(* CoDeSys 2.3 export: 6SHU-P2_V2.EXP *)

(* POU MAIN, CFC *)
PROGRAM MAIN
VAR
	TCT: ISTOK_TaskCycleTime;
END_VAR
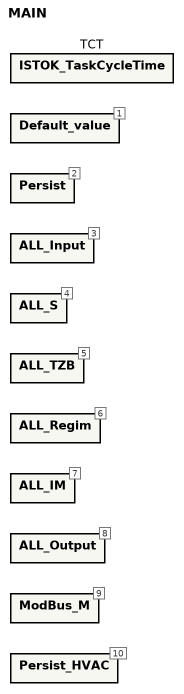
_CFC_ (* Continuous Function Chart, elements in execution order *)
#0 TCT:ISTOK_TaskCycleTime()
#1 Default_value()
#2 Persist()
#3 ALL_Input()
#4 ALL_S()
#5 ALL_TZB()
#6 ALL_Regim()
#7 ALL_IM()
#8 ALL_Output()
#9 ModBus_M()
#10 Persist_HVAC()
_END_CFC_
(* the same logic as Structured Text *)
TCT();
Default_value();
Persist();
ALL_Input();
ALL_S();
ALL_TZB();
ALL_Regim();
ALL_IM();
ALL_Output();
ModBus_M();
Persist_HVAC();
END_PROGRAM

(* POU Lib/ISTOK_TaskCycleTime, CFC *)
FUNCTION_BLOCK ISTOK_TaskCycleTime
VAR_INPUT
END_VAR
VAR_OUTPUT
END_VAR
VAR
END_VAR
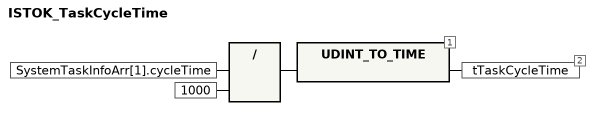
_CFC_ (* Continuous Function Chart, elements in execution order *)
#0 /(SystemTaskInfoArr[1].cycleTime, 1000)
#1 UDINT_TO_TIME(#0)
#2 tTaskCycleTime <= #1
_END_CFC_
END_FUNCTION_BLOCK

(* POU Default_value, CFC *)
PROGRAM Default_value
VAR
END_VAR
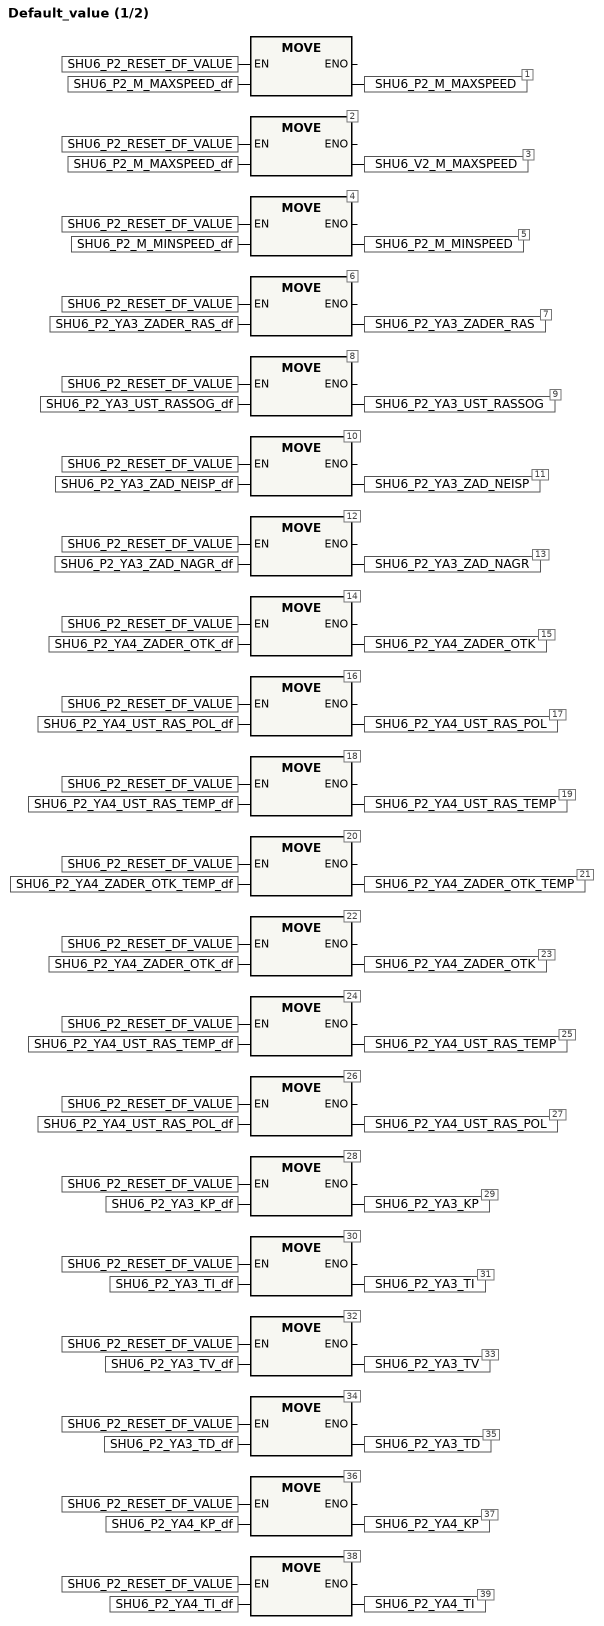
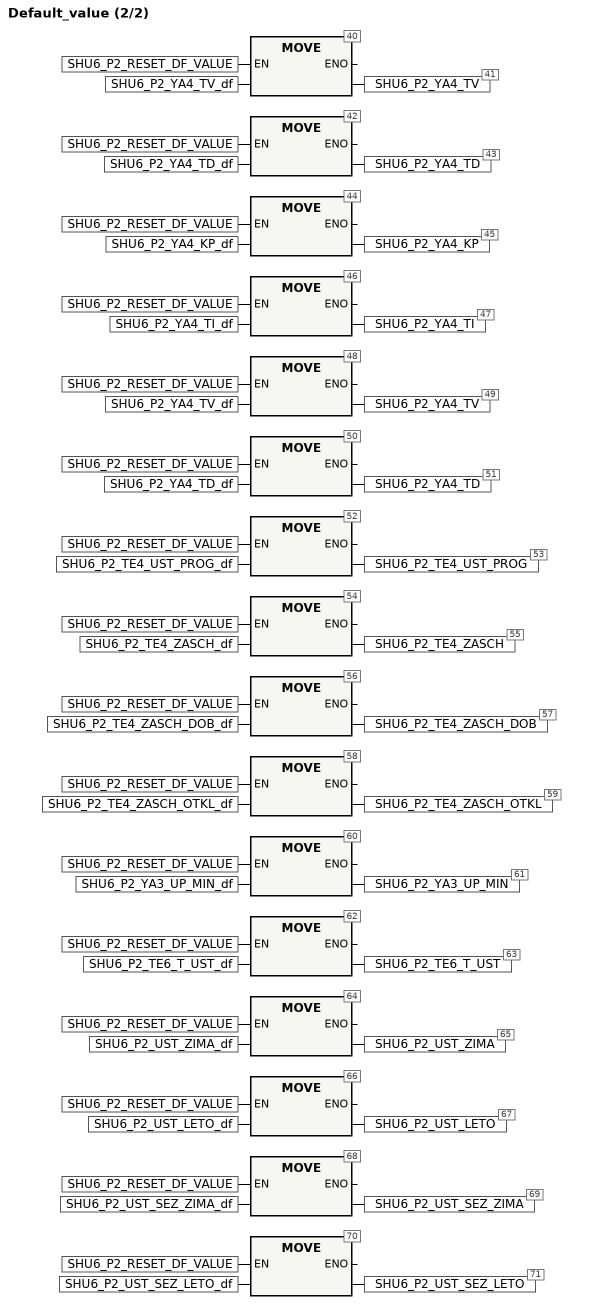
_CFC_ (* Continuous Function Chart, elements in execution order *)
#0 MOVE(EN: SHU6_P2_RESET_DF_VALUE, SHU6_P2_M_MAXSPEED_df)
#1 SHU6_P2_M_MAXSPEED <= #0
#2 MOVE(EN: SHU6_P2_RESET_DF_VALUE, SHU6_P2_M_MAXSPEED_df)
#3 SHU6_V2_M_MAXSPEED <= #2
#4 MOVE(EN: SHU6_P2_RESET_DF_VALUE, SHU6_P2_M_MINSPEED_df)
#5 SHU6_P2_M_MINSPEED <= #4
#6 MOVE(EN: SHU6_P2_RESET_DF_VALUE, SHU6_P2_YA3_ZADER_RAS_df)
#7 SHU6_P2_YA3_ZADER_RAS <= #6
#8 MOVE(EN: SHU6_P2_RESET_DF_VALUE, SHU6_P2_YA3_UST_RASSOG_df)
#9 SHU6_P2_YA3_UST_RASSOG <= #8
#10 MOVE(EN: SHU6_P2_RESET_DF_VALUE, SHU6_P2_YA3_ZAD_NEISP_df)
#11 SHU6_P2_YA3_ZAD_NEISP <= #10
#12 MOVE(EN: SHU6_P2_RESET_DF_VALUE, SHU6_P2_YA3_ZAD_NAGR_df)
#13 SHU6_P2_YA3_ZAD_NAGR <= #12
#14 MOVE(EN: SHU6_P2_RESET_DF_VALUE, SHU6_P2_YA4_ZADER_OTK_df)
#15 SHU6_P2_YA4_ZADER_OTK <= #14
#16 MOVE(EN: SHU6_P2_RESET_DF_VALUE, SHU6_P2_YA4_UST_RAS_POL_df)
#17 SHU6_P2_YA4_UST_RAS_POL <= #16
#18 MOVE(EN: SHU6_P2_RESET_DF_VALUE, SHU6_P2_YA4_UST_RAS_TEMP_df)
#19 SHU6_P2_YA4_UST_RAS_TEMP <= #18
#20 MOVE(EN: SHU6_P2_RESET_DF_VALUE, SHU6_P2_YA4_ZADER_OTK_TEMP_df)
#21 SHU6_P2_YA4_ZADER_OTK_TEMP <= #20
#22 MOVE(EN: SHU6_P2_RESET_DF_VALUE, SHU6_P2_YA4_ZADER_OTK_df)
#23 SHU6_P2_YA4_ZADER_OTK <= #22
#24 MOVE(EN: SHU6_P2_RESET_DF_VALUE, SHU6_P2_YA4_UST_RAS_TEMP_df)
#25 SHU6_P2_YA4_UST_RAS_TEMP <= #24
#26 MOVE(EN: SHU6_P2_RESET_DF_VALUE, SHU6_P2_YA4_UST_RAS_POL_df)
#27 SHU6_P2_YA4_UST_RAS_POL <= #26
#28 MOVE(EN: SHU6_P2_RESET_DF_VALUE, SHU6_P2_YA3_KP_df)
#29 SHU6_P2_YA3_KP <= #28
#30 MOVE(EN: SHU6_P2_RESET_DF_VALUE, SHU6_P2_YA3_TI_df)
#31 SHU6_P2_YA3_TI <= #30
#32 MOVE(EN: SHU6_P2_RESET_DF_VALUE, SHU6_P2_YA3_TV_df)
#33 SHU6_P2_YA3_TV <= #32
#34 MOVE(EN: SHU6_P2_RESET_DF_VALUE, SHU6_P2_YA3_TD_df)
#35 SHU6_P2_YA3_TD <= #34
#36 MOVE(EN: SHU6_P2_RESET_DF_VALUE, SHU6_P2_YA4_KP_df)
#37 SHU6_P2_YA4_KP <= #36
#38 MOVE(EN: SHU6_P2_RESET_DF_VALUE, SHU6_P2_YA4_TI_df)
#39 SHU6_P2_YA4_TI <= #38
#40 MOVE(EN: SHU6_P2_RESET_DF_VALUE, SHU6_P2_YA4_TV_df)
#41 SHU6_P2_YA4_TV <= #40
#42 MOVE(EN: SHU6_P2_RESET_DF_VALUE, SHU6_P2_YA4_TD_df)
#43 SHU6_P2_YA4_TD <= #42
#44 MOVE(EN: SHU6_P2_RESET_DF_VALUE, SHU6_P2_YA4_KP_df)
#45 SHU6_P2_YA4_KP <= #44
#46 MOVE(EN: SHU6_P2_RESET_DF_VALUE, SHU6_P2_YA4_TI_df)
#47 SHU6_P2_YA4_TI <= #46
#48 MOVE(EN: SHU6_P2_RESET_DF_VALUE, SHU6_P2_YA4_TV_df)
#49 SHU6_P2_YA4_TV <= #48
#50 MOVE(EN: SHU6_P2_RESET_DF_VALUE, SHU6_P2_YA4_TD_df)
#51 SHU6_P2_YA4_TD <= #50
#52 MOVE(EN: SHU6_P2_RESET_DF_VALUE, SHU6_P2_TE4_UST_PROG_df)
#53 SHU6_P2_TE4_UST_PROG <= #52
#54 MOVE(EN: SHU6_P2_RESET_DF_VALUE, SHU6_P2_TE4_ZASCH_df)
#55 SHU6_P2_TE4_ZASCH <= #54
#56 MOVE(EN: SHU6_P2_RESET_DF_VALUE, SHU6_P2_TE4_ZASCH_DOB_df)
#57 SHU6_P2_TE4_ZASCH_DOB <= #56
#58 MOVE(EN: SHU6_P2_RESET_DF_VALUE, SHU6_P2_TE4_ZASCH_OTKL_df)
#59 SHU6_P2_TE4_ZASCH_OTKL <= #58
#60 MOVE(EN: SHU6_P2_RESET_DF_VALUE, SHU6_P2_YA3_UP_MIN_df)
#61 SHU6_P2_YA3_UP_MIN <= #60
#62 MOVE(EN: SHU6_P2_RESET_DF_VALUE, SHU6_P2_TE6_T_UST_df)
#63 SHU6_P2_TE6_T_UST <= #62
#64 MOVE(EN: SHU6_P2_RESET_DF_VALUE, SHU6_P2_UST_ZIMA_df)
#65 SHU6_P2_UST_ZIMA <= #64
#66 MOVE(EN: SHU6_P2_RESET_DF_VALUE, SHU6_P2_UST_LETO_df)
#67 SHU6_P2_UST_LETO <= #66
#68 MOVE(EN: SHU6_P2_RESET_DF_VALUE, SHU6_P2_UST_SEZ_ZIMA_df)
#69 SHU6_P2_UST_SEZ_ZIMA <= #68
#70 MOVE(EN: SHU6_P2_RESET_DF_VALUE, SHU6_P2_UST_SEZ_LETO_df)
#71 SHU6_P2_UST_SEZ_LETO <= #70
_END_CFC_
(* the same logic as Structured Text *)
IF SHU6_P2_RESET_DF_VALUE THEN SHU6_P2_M_MAXSPEED := SHU6_P2_M_MAXSPEED_df; END_IF;
IF SHU6_P2_RESET_DF_VALUE THEN SHU6_V2_M_MAXSPEED := SHU6_P2_M_MAXSPEED_df; END_IF;
IF SHU6_P2_RESET_DF_VALUE THEN SHU6_P2_M_MINSPEED := SHU6_P2_M_MINSPEED_df; END_IF;
IF SHU6_P2_RESET_DF_VALUE THEN SHU6_P2_YA3_ZADER_RAS := SHU6_P2_YA3_ZADER_RAS_df; END_IF;
IF SHU6_P2_RESET_DF_VALUE THEN SHU6_P2_YA3_UST_RASSOG := SHU6_P2_YA3_UST_RASSOG_df; END_IF;
IF SHU6_P2_RESET_DF_VALUE THEN SHU6_P2_YA3_ZAD_NEISP := SHU6_P2_YA3_ZAD_NEISP_df; END_IF;
IF SHU6_P2_RESET_DF_VALUE THEN SHU6_P2_YA3_ZAD_NAGR := SHU6_P2_YA3_ZAD_NAGR_df; END_IF;
IF SHU6_P2_RESET_DF_VALUE THEN SHU6_P2_YA4_ZADER_OTK := SHU6_P2_YA4_ZADER_OTK_df; END_IF;
IF SHU6_P2_RESET_DF_VALUE THEN SHU6_P2_YA4_UST_RAS_POL := SHU6_P2_YA4_UST_RAS_POL_df; END_IF;
IF SHU6_P2_RESET_DF_VALUE THEN SHU6_P2_YA4_UST_RAS_TEMP := SHU6_P2_YA4_UST_RAS_TEMP_df; END_IF;
IF SHU6_P2_RESET_DF_VALUE THEN SHU6_P2_YA4_ZADER_OTK_TEMP := SHU6_P2_YA4_ZADER_OTK_TEMP_df; END_IF;
IF SHU6_P2_RESET_DF_VALUE THEN SHU6_P2_YA4_ZADER_OTK := SHU6_P2_YA4_ZADER_OTK_df; END_IF;
IF SHU6_P2_RESET_DF_VALUE THEN SHU6_P2_YA4_UST_RAS_TEMP := SHU6_P2_YA4_UST_RAS_TEMP_df; END_IF;
IF SHU6_P2_RESET_DF_VALUE THEN SHU6_P2_YA4_UST_RAS_POL := SHU6_P2_YA4_UST_RAS_POL_df; END_IF;
IF SHU6_P2_RESET_DF_VALUE THEN SHU6_P2_YA3_KP := SHU6_P2_YA3_KP_df; END_IF;
IF SHU6_P2_RESET_DF_VALUE THEN SHU6_P2_YA3_TI := SHU6_P2_YA3_TI_df; END_IF;
IF SHU6_P2_RESET_DF_VALUE THEN SHU6_P2_YA3_TV := SHU6_P2_YA3_TV_df; END_IF;
IF SHU6_P2_RESET_DF_VALUE THEN SHU6_P2_YA3_TD := SHU6_P2_YA3_TD_df; END_IF;
IF SHU6_P2_RESET_DF_VALUE THEN SHU6_P2_YA4_KP := SHU6_P2_YA4_KP_df; END_IF;
IF SHU6_P2_RESET_DF_VALUE THEN SHU6_P2_YA4_TI := SHU6_P2_YA4_TI_df; END_IF;
IF SHU6_P2_RESET_DF_VALUE THEN SHU6_P2_YA4_TV := SHU6_P2_YA4_TV_df; END_IF;
IF SHU6_P2_RESET_DF_VALUE THEN SHU6_P2_YA4_TD := SHU6_P2_YA4_TD_df; END_IF;
IF SHU6_P2_RESET_DF_VALUE THEN SHU6_P2_YA4_KP := SHU6_P2_YA4_KP_df; END_IF;
IF SHU6_P2_RESET_DF_VALUE THEN SHU6_P2_YA4_TI := SHU6_P2_YA4_TI_df; END_IF;
IF SHU6_P2_RESET_DF_VALUE THEN SHU6_P2_YA4_TV := SHU6_P2_YA4_TV_df; END_IF;
IF SHU6_P2_RESET_DF_VALUE THEN SHU6_P2_YA4_TD := SHU6_P2_YA4_TD_df; END_IF;
IF SHU6_P2_RESET_DF_VALUE THEN SHU6_P2_TE4_UST_PROG := SHU6_P2_TE4_UST_PROG_df; END_IF;
IF SHU6_P2_RESET_DF_VALUE THEN SHU6_P2_TE4_ZASCH := SHU6_P2_TE4_ZASCH_df; END_IF;
IF SHU6_P2_RESET_DF_VALUE THEN SHU6_P2_TE4_ZASCH_DOB := SHU6_P2_TE4_ZASCH_DOB_df; END_IF;
IF SHU6_P2_RESET_DF_VALUE THEN SHU6_P2_TE4_ZASCH_OTKL := SHU6_P2_TE4_ZASCH_OTKL_df; END_IF;
IF SHU6_P2_RESET_DF_VALUE THEN SHU6_P2_YA3_UP_MIN := SHU6_P2_YA3_UP_MIN_df; END_IF;
IF SHU6_P2_RESET_DF_VALUE THEN SHU6_P2_TE6_T_UST := SHU6_P2_TE6_T_UST_df; END_IF;
IF SHU6_P2_RESET_DF_VALUE THEN SHU6_P2_UST_ZIMA := SHU6_P2_UST_ZIMA_df; END_IF;
IF SHU6_P2_RESET_DF_VALUE THEN SHU6_P2_UST_LETO := SHU6_P2_UST_LETO_df; END_IF;
IF SHU6_P2_RESET_DF_VALUE THEN SHU6_P2_UST_SEZ_ZIMA := SHU6_P2_UST_SEZ_ZIMA_df; END_IF;
IF SHU6_P2_RESET_DF_VALUE THEN SHU6_P2_UST_SEZ_LETO := SHU6_P2_UST_SEZ_LETO_df; END_IF;
END_PROGRAM

(* POU Persist, ST *)
PROGRAM Persist
VAR
	Save: WritePersistentData;
END_VAR
Save(NETID:='10.150.4.62.1.1',PORT:=801,START:=TRUE,TMOUT:=t#1s ,BUSY=> ,ERR=> ,	ERRID=> );
Save(NETID:='10.150.4.62.1.1',PORT:=801,START:= FALSE ,TMOUT:=t#1s ,BUSY=> ,ERR=> ,ERRID=> );
END_PROGRAM

(* POU Input/ALL_Input, CFC *)
PROGRAM ALL_Input
VAR
END_VAR
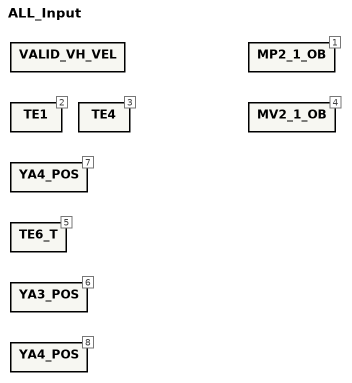
_CFC_ (* Continuous Function Chart, elements in execution order *)
#0 VALID_VH_VEL()
#1 MP2_1_OB()
#2 TE1()
#3 TE4()
#4 MV2_1_OB()
#5 TE6_T()
#6 YA3_POS()
#7 YA4_POS()
#8 YA4_POS()
_END_CFC_
(* the same logic as Structured Text *)
VALID_VH_VEL();
MP2_1_OB();
TE1();
TE4();
MV2_1_OB();
TE6_T();
YA3_POS();
YA4_POS();
YA4_POS();
END_PROGRAM

(* POU Input/VALID_VH_VEL, CFC *)
PROGRAM VALID_VH_VEL
VAR
	SHU6_P2_UST_SEZ_LETO_OLD: REAL;
	SHU6_P2_UST_SEZ_ZIMA_OLD: REAL;

	RT_VKL_OLD_SEZ_LETO: R_TRIG;
	RT_VKL_OLD_SEZ_ZIMA: R_TRIG;

	(*_____________________________________*)
	SHU6_P2_UE1_VL_UST_OTKL_OLD: REAL;
	SHU6_P2_UE1_VL_UST_VKL_OLD: REAL;

	RT_TE6_VL_UST_OTKL_OLD: R_TRIG;
	RT_TE6_VL_UST_VKL_OLD: R_TRIG;

	(*_____________________________________*)
	RT_UE3_VL_UST_OTKL_OLD: R_TRIG;
	RT_UE3_VL_UST_VKL_OLD: R_TRIG;
	SHU6_P2_TE6_VL_UST_OTKL_OLD: REAL;
	SHU6_P2_TE6_VL_UST_VKL_OLD: REAL;

	(*_____________________________________*)
	RT_TE6_TE_UST_OTKL_OLD: R_TRIG;
	RT_UE3_TE_UST_VKL_OLD: R_TRIG;

	SHU6_P2_UE1_T_UST_OLD: REAL;
	SHU6_P2_TE6_T_UST_OLD: REAL;
END_VAR
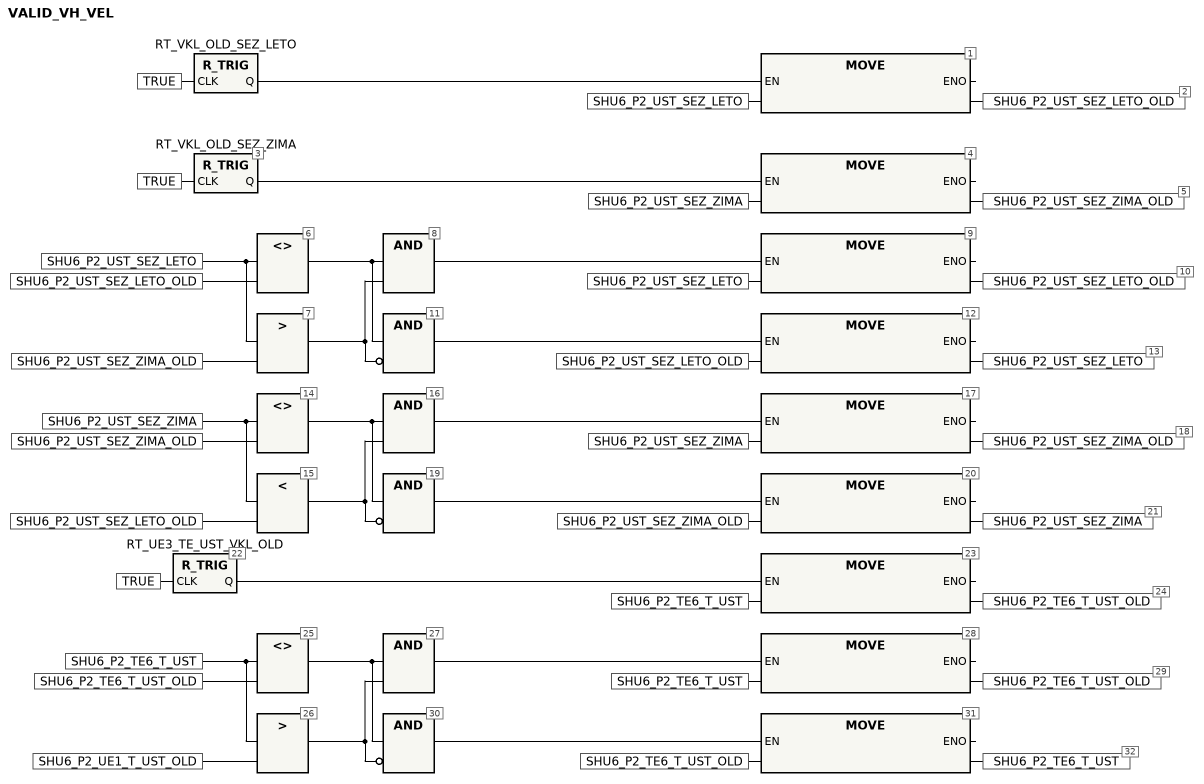
